// TIA Portal V17 export
// export: Created 2024-01-30T08:49:15.9939561Z, ExportSetting WithDefaults, DisplayName Totally Integrated Automation Portal, DisplayVersion V17 Update 6, DisplayName TIA Portal Openness, DisplayVersion V17 Update 6, DisplayName TIA Portal Version Control Interface, DisplayVersion V17, DisplayName STEP 7 Professional, DisplayVersion V17 Update 6, DisplayName STEP 7 Safety, DisplayVersion V17 Update 6, DisplayName WinCC Advanced, DisplayVersion V17 Update 6
FUNCTION_BLOCK "FB_DATA_LOGGING"   // FB13, LAD
{ S7_Optimized_Access := 'TRUE' }
VERSION : 0.1
// stored: AutoNumber true, IsIECCheckEnabled false, IsRetainMemResEnabled false, MemoryReserve 100, SetENOAutomatically false, UDAEnableTagReadback false
   VAR
      DataLogCreate_Instance { S7_SetPoint := 'True'} : DataLogCreate;
      DataLogWrite_Instance { S7_SetPoint := 'True'} : DataLogWrite;
      DataLogNewFile_Instance { S7_SetPoint := 'True'} : DataLogNewFile;
      DataLogNewFile_Instance_1 { S7_SetPoint := 'True'} : DataLogNewFile;
      DataLogDelete_Instance { S7_SetPoint := 'True'} : DataLogDelete;
      DataLogClear_Instance { S7_SetPoint := 'True'} : DataLogClear;
   END_VAR
BEGIN

REGION Network 1: Data Log Create
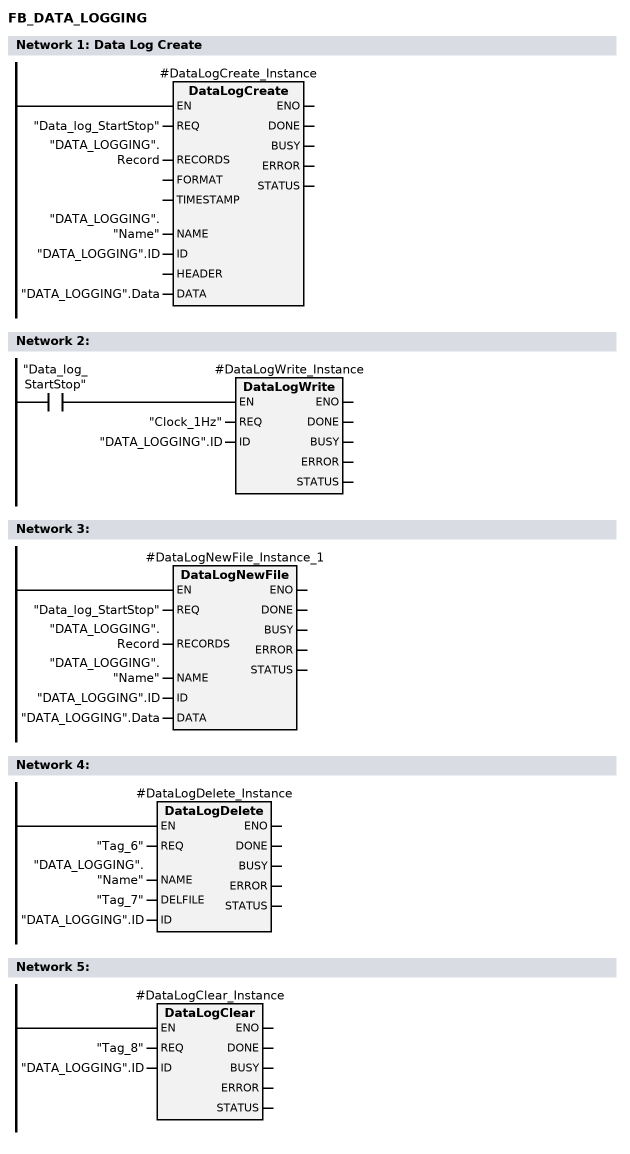
   RUNG wire#powerrail
      #DataLogCreate_Instance.DataLogCreate(REQ := "Data_log_StartStop", RECORDS := "DATA_LOGGING".Record, FORMAT :=, TIMESTAMP :=, "NAME" := "DATA_LOGGING"."Name", ID := "DATA_LOGGING".ID, HEADER :=, DATA := "DATA_LOGGING".Data, DONE =>, BUSY =>, ERROR =>, STATUS =>)
   END_RUNG
   // the same network as SCL:
   #DataLogCreate_Instance(REQ := "Data_log_StartStop",   // DataLogCreate
                           RECORDS := "DATA_LOGGING".Record,
                           "NAME" := "DATA_LOGGING"."Name",
                           ID := "DATA_LOGGING".ID,
                           DATA := "DATA_LOGGING".Data);
END_REGION

REGION Network 2
   RUNG wire#powerrail
      Contact( "Data_log_StartStop" )
      #DataLogWrite_Instance.DataLogWrite(REQ := "Clock_1Hz", ID := "DATA_LOGGING".ID, DONE =>, BUSY =>, ERROR =>, STATUS =>)
   END_RUNG
   // the same network as SCL:
   IF "Data_log_StartStop" THEN
       #DataLogWrite_Instance(REQ := "Clock_1Hz", ID := "DATA_LOGGING".ID);   // DataLogWrite
   END_IF;
END_REGION

REGION Network 3
   RUNG wire#powerrail
      { S7_Templates := "card := 1" } #DataLogNewFile_Instance_1.DataLogNewFile(REQ := "Data_log_StartStop", RECORDS := "DATA_LOGGING".Record, "NAME" := "DATA_LOGGING"."Name", ID := "DATA_LOGGING".ID, Data := "DATA_LOGGING".Data, DONE =>, BUSY =>, ERROR =>, STATUS =>)
   END_RUNG
   // the same network as SCL:
   #DataLogNewFile_Instance_1(REQ := "Data_log_StartStop",   // DataLogNewFile
                           RECORDS := "DATA_LOGGING".Record,
                           "NAME" := "DATA_LOGGING"."Name",
                           ID := "DATA_LOGGING".ID,
                           Data := "DATA_LOGGING".Data);
END_REGION

REGION Network 4
   RUNG wire#powerrail
      #DataLogDelete_Instance.DataLogDelete(REQ := "Tag_6", "NAME" := "DATA_LOGGING"."Name", DelFile := "Tag_7", ID := "DATA_LOGGING".ID, DONE =>, BUSY =>, ERROR =>, STATUS =>)
   END_RUNG
   // the same network as SCL:
   #DataLogDelete_Instance(REQ := "Tag_6",   // DataLogDelete
                           "NAME" := "DATA_LOGGING"."Name",
                           DelFile := "Tag_7",
                           ID := "DATA_LOGGING".ID);
END_REGION

REGION Network 5
   RUNG wire#powerrail
      #DataLogClear_Instance.DataLogClear(REQ := "Tag_8", ID := "DATA_LOGGING".ID, DONE =>, BUSY =>, ERROR =>, STATUS =>)
   END_RUNG
   // the same network as SCL:
   #DataLogClear_Instance(REQ := "Tag_8", ID := "DATA_LOGGING".ID);   // DataLogClear
END_REGION
END_FUNCTION_BLOCK
